// Block: PPrgArchive11

DATA_BLOCK PPrgArchive11
VERSION : 0.1
   NON_RETAIN
   VAR
      PRG : Array[1001..1100] of PPrg_Data;
   END_VAR

BEGIN
   // No initialization required
END_DATA_BLOCK
